FUNCTION_BLOCK FlushSludgeBufferCond (* Basic Function Block Type *)
  (* Standard: 61499-2 *)
  (* Version 0.0, 5/26/2024, SESA713705, Schneider Electric, Template *)
  PACKAGE SE.Nereda;
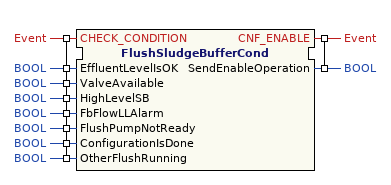
  EVENT_INPUT
    CHECK_CONDITION WITH EffluentLevelIsOK, FbFlowLLAlarm, ValveAvailable, ConfigurationIsDone, FlushPumpNotReady, HighLevelSB, OtherFlushRunning;
  END_EVENT
  EVENT_OUTPUT
    CNF_ENABLE WITH SendEnableOperation;
  END_EVENT
  VAR_INPUT
    EffluentLevelIsOK : BOOL;
    ValveAvailable : BOOL;
    HighLevelSB : BOOL;
    FbFlowLLAlarm : BOOL;
    FlushPumpNotReady : BOOL;
    ConfigurationIsDone : BOOL;
    OtherFlushRunning : BOOL;
  END_VAR
  VAR_OUTPUT
    SendEnableOperation : BOOL;
  END_VAR
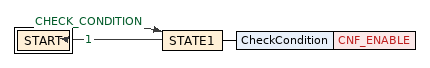
  EC_STATES
    START; (* Initial State *)
    STATE1 : CheckCondition -> CNF_ENABLE;
  END_STATES
  EC_TRANSITIONS
    START TO STATE1 := CHECK_CONDITION;
    STATE1 TO START := 1;
  END_TRANSITIONS
  ALGORITHM CheckCondition IN ST:
;
IF 	EffluentLevelIsOK AND
	NOT FbFlowLLAlarm AND
	ValveAvailable AND
	NOT HighLevelSB AND
	NOT FlushPumpNotReady AND
	NOT OtherFlushRunning AND
	ConfigurationIsDone	THEN

	SendEnableOperation := TRUE;
ELSE
	SendEnableOperation := FALSE;
END_IF;
  END_ALGORITHM
END_FUNCTION_BLOCK
